// TIA Portal V21 export
TYPE "ElencoCampionature"
   STRUCT
      h { S7_SetPoint := 'True'} : Array[1..24] of "Campionatura";
   END_STRUCT;
END_TYPE
